// TIA Portal V19 export
FUNCTION "ToDo" : Void   // FC999, STL
{ S7_Optimized_Access := 'FALSE' }
// stored: AutoNumber false
BEGIN

NETWORK
TITLE = 
      CLR;
      L     0;

END_FUNCTION
